FUNCTION_BLOCK E_TimeOut (* Simple implementation of the timeout services *)
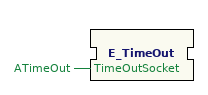
  SOCKETS
    TimeOutSocket : iec61499::events::ATimeOut;
  END_SOCKETS
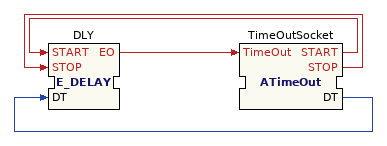
  FBS
    DLY : iec61499::events::E_DELAY;
  END_FBS
  EVENT_CONNECTIONS
    TimeOutSocket.START TO DLY.START;
    TimeOutSocket.STOP TO DLY.STOP;
    DLY.EO TO TimeOutSocket.TimeOut;
  END_CONNECTIONS
  DATA_CONNECTIONS
    TimeOutSocket.DT TO DLY.DT;
  END_CONNECTIONS
END_FUNCTION_BLOCK
